Staubli VAL3: test_ventouse.pgx

program test_ventouse()
begin
  movej(jP1, ventouse, mNomSpeed)
  movej(jP2, ventouse, mNomSpeed)
  doValve1=true
  movej(jP4, ventouse, mNomSpeed)
  movej(jP5, ventouse, mNomSpeed)
  movej(jP3, ventouse, mNomSpeed)
  doValve1=false
  movej(jP1, ventouse, mNomSpeed)
  movej(jP3, ventouse, mNomSpeed)
  doValve1=true
  movej(jP5, ventouse, mNomSpeed)
  movej(jP4, ventouse, mNomSpeed)
  movej(jP2, ventouse, mNomSpeed)
  doValve1=true
  waitEndMove()
end
